FUNCTION_BLOCK FB_PressedButton
VAR_INPUT
	bIsButtonPressed : BOOL;
END_VAR
VAR_OUTPUT
	bLightOfPressedButton : BOOL;
END_VAR
VAR
END_VAR

// As long as the button is pressed the light is on, when it's not pressed, light turns off
IF bIsButtonPressed THEN
	bLightOfPressedButton := TRUE;
ELSE
	bLightOfPressedButton := FALSE;
END_IF

END_FUNCTION_BLOCK

(* stored: Version 1.1.0.1, ProductVersion 3.1.4024.12
   POU FB_PressedButton: Id {ba9c4601-6d6c-4137-b66e-50138fd94acc}, SpecialFunc None *)
